(* PLC project autom_ihm_rmll, lolitech autom_ihm_rmll 1 *)
(* stored: creationDateTime 2008-06-28 15:43:31, modificationDateTime 2008-06-28 18:26:40 *)

FUNCTION_BLOCK automate
  VAR_OUTPUT
    pump : BOOL;
    sink : BOOL;
  END_VAR
  VAR_INPUT
    do_empty : BOOL;
    do_fill : BOOL;
    full : BOOL;
    empty : BOOL;
  END_VAR
  VAR  (* added by the conversion: wires and edge detectors of the diagram *)
    _AND19_OUT : BOOL;
  END_VAR

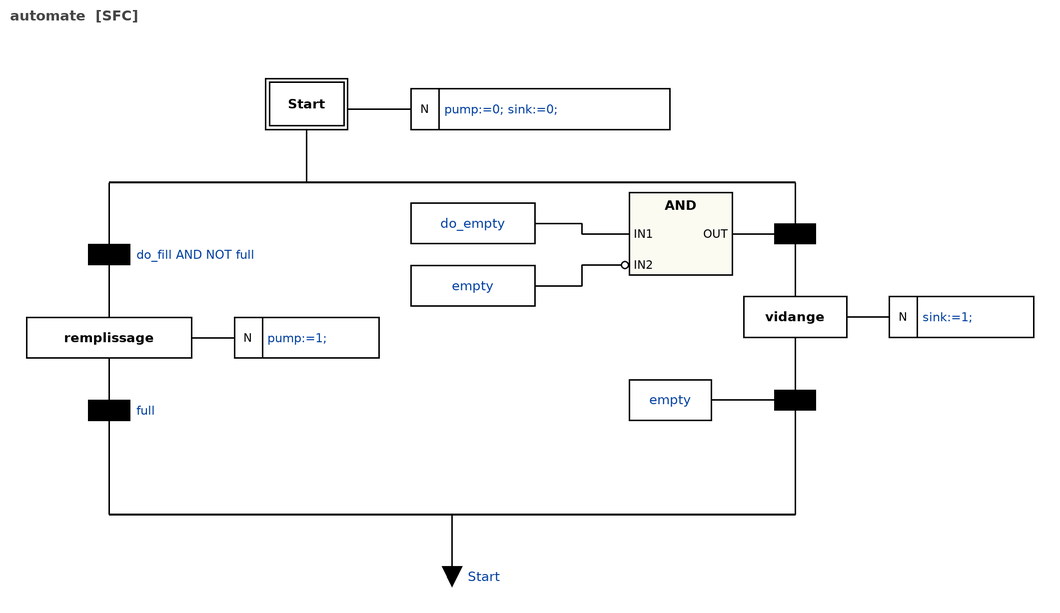
INITIAL_STEP Start:
  START_INLINE1(N);
  COMPUTE_FUNCTION_BLOCKS(S);
END_STEP
ACTION START_INLINE1:
  pump:=0; sink:=0;
END_ACTION
TRANSITION FROM Start TO vidange
  := _AND19_OUT;
END_TRANSITION
TRANSITION FROM Start TO remplissage
  := do_fill AND NOT full;
END_TRANSITION
STEP vidange:
  VIDANGE_INLINE2(N);
END_STEP
ACTION VIDANGE_INLINE2:
  sink:=1;
END_ACTION
TRANSITION FROM vidange TO Start
  := empty;
END_TRANSITION
STEP remplissage:
  REMPLISSAGE_INLINE3(N);
END_STEP
ACTION REMPLISSAGE_INLINE3:
  pump:=1;
END_ACTION
TRANSITION FROM remplissage TO Start
  := full;
END_TRANSITION
ACTION COMPUTE_FUNCTION_BLOCKS:  (* blocks drawn on the SFC sheet *)
  _AND19_OUT := do_empty AND NOT empty;
END_ACTION
END_FUNCTION_BLOCK

FUNCTION_BLOCK control_gauge
  VAR_INPUT
    Xin : REAL;
    Yin : REAL;
  END_VAR
  VAR_OUTPUT
    Xout : REAL;
    Yout : REAL;
  END_VAR
  VAR_INPUT
    Consigne : INT;
  END_VAR
  VAR
    Initialized : BOOL := false;
    Xtmp : REAL;
    Ytmp : REAL;
  END_VAR

IF NOT INITIALIZED THEN
  XTMP := XIN;
  YTMP := YIN;
  INITIALIZED := TRUE;
END_IF;
XOUT := XTMP * INT_TO_REAL(CONSIGNE) / 100.0;
YOUT := YTMP * INT_TO_REAL(CONSIGNE) / 100.0;
          
END_FUNCTION_BLOCK

PROGRAM main
  VAR
    ctrl_gauge1 : control_gauge;
    fill : Button;
    empty : Button;
    gauge : Transform;
  END_VAR
  VAR
    level AT %IW1.0.3.8196.0 : INT;
    pump_out AT %QX1.0.3.8192.0 : BOOL;
    sink_out AT %QX1.0.3.8193.0 : BOOL;
    full_in AT %IX1.0.3.8194.0 : BOOL;
    empty_in AT %IX1.0.3.8195.0 : BOOL;
  END_VAR
  VAR
    controleur : automate;
  END_VAR

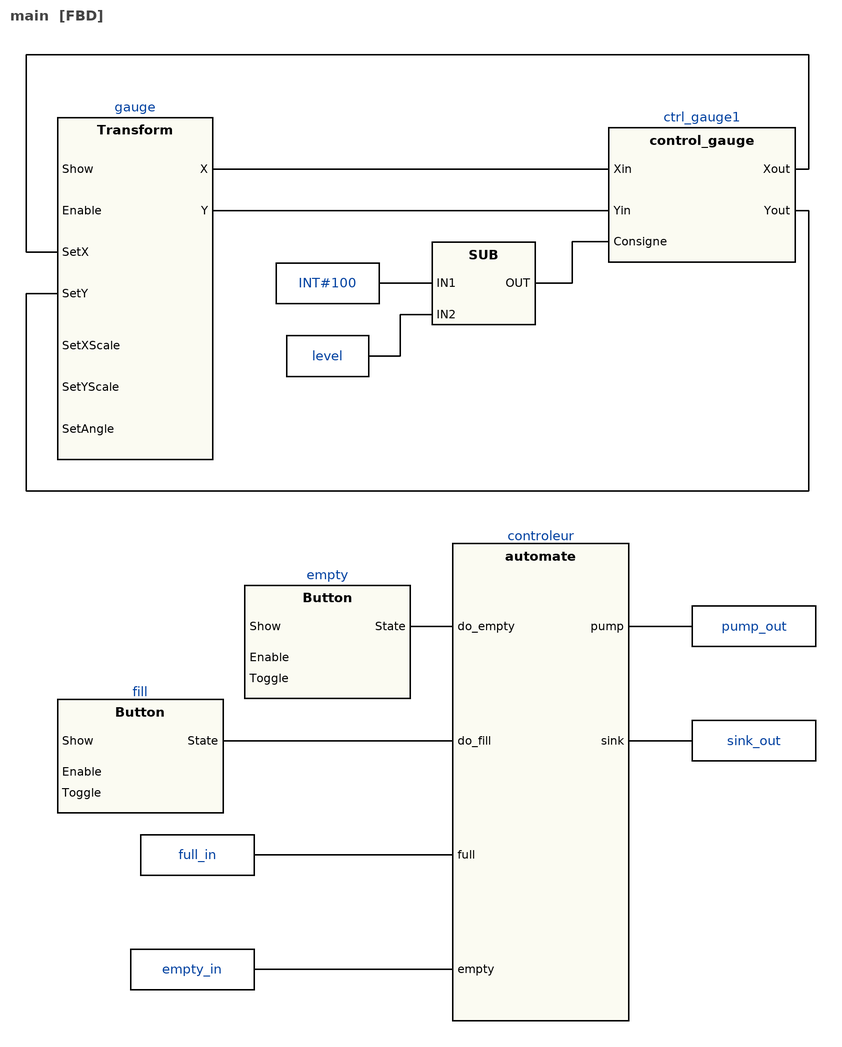
(* FBD diagram, written out as Structured Text *)
empty();
fill();
controleur(do_empty := empty.State, do_fill := fill.State, full := full_in, empty := empty_in);
pump_out := controleur.pump;
sink_out := controleur.sink;
ctrl_gauge1(Xin := gauge.X, Yin := gauge.Y, Consigne := INT#100 - level);
gauge(SetX := ctrl_gauge1.Xout, SetY := ctrl_gauge1.Yout);
END_PROGRAM

CONFIGURATION conf
  RESOURCE ress ON PLC
    TASK matache(INTERVAL := 00:00:00.100000, PRIORITY := 0);
    PROGRAM moninst WITH matache : main;
  END_RESOURCE
END_CONFIGURATION
